// Feedback 2 gear denominator
TYPE ST_P183 :
STRUCT
	Feedback_2_geat_denominator:UDINT;
END_STRUCT
END_TYPE

(* stored: Version 1.1.0.1, ProductVersion 3.1.4024.6
   DUT ST_P183: Id {3c7eb6d6-56ef-4dbb-9b9b-f618e4ddfe95} *)
